{attribute 'no_explicit_call' := 'do not call this function block directly'} 
{attribute 'enable_dynamic_creation'}
FUNCTION_BLOCK ListOfBytesEnumerator EXTENDS PointerBasedEnumerator
VAR
	_ClassName : STRING := __POUNAME();
	_List : IReadOnlyListOfBytes;
	_Current : POINTER TO BYTE;
END_VAR

{attribute 'monitoring' := 'call'}
PROPERTY ClassName : STRING
GET
ClassName := _ClassName;
END_GET
END_PROPERTY

{attribute 'OPC.UA.DA.Property' := '1'}
{attribute 'monitoring' := 'call'}
PROPERTY Current : PVOID
GET
Current := _Current;
END_GET
END_PROPERTY

METHOD INTERNAL Initialize
VAR_INPUT
	list : IReadOnlyListOfBytes;
END_VAR
_List := list;
END_METHOD

{attribute "object_name" := "MoveNext"}
METHOD MoveNext : BOOL
_CurrentIndex := _CurrentIndex + 1;	

IF _CurrentIndex >= _List.Count THEN
	_Current := 0;
	_CurrentIndex := _List.Count;
ELSE
	_Current := _List.Get(_CurrentIndex);	
	MoveNext := TRUE;
END_IF
END_METHOD

{attribute "object_name" := "Reset"}
METHOD Reset
SUPER^.Reset();

_Current := 0;
END_METHOD

{attribute 'monitoring' := 'call'}
PROPERTY Size : ULINT
GET
Size := XSIZEOF(THIS^);
END_GET
END_PROPERTY

END_FUNCTION_BLOCK

(* stored: Version 1.1.0.1
   POU ListOfBytesEnumerator: Id {e5f28ca5-1848-0aab-3385-3fb94b3f640c}, SpecialFunc None
   Property ClassName: Id {89e1bb34-f534-0ed0-3918-be98a7eb3011}
   Get Get: Id {a92920f3-3ce7-03e7-3445-0b1ae94b6b28}
   Property Current: Id {90f7e8b1-5b06-06eb-1be9-fba8f1e6a61d}
   Get Get: Id {936ecc96-a4c7-0bc6-2af0-ec01eb201e13}
   Method Initialize: Id {7065af19-d111-0b51-0461-9593ca28feaf}
   Method MoveNext: Id {b1fe29f1-4d65-0b4b-2b56-632a8663a457}
   Method Reset: Id {8c897b44-69bf-040e-3585-fd89874c3015}
   Property Size: Id {b05b8dcf-1356-4ef5-977c-d0b3f241e80e}
   Get Get: Id {38c1b824-501f-4f6e-af69-41fbb7a3b874} *)
